// TIA Portal V17 export
// export: Created 2023-02-26T22:53:27.9284899Z, ExportSetting WithDefaults, DisplayName Totally Integrated Automation Portal, DisplayVersion V17, DisplayName TIA Portal Openness, DisplayVersion V17, DisplayName TIA Portal Version Control Interface, DisplayVersion V17, DisplayName TIA Portal Test Suite Advanced, DisplayVersion V17, DisplayName STEP 7 Professional, DisplayVersion V17, DisplayName SIMATIC Energy Suite, DisplayVersion V17, DisplayName STEP 7 Safety, DisplayVersion V17, DisplayName WinCC Professional, DisplayVersion V17
FUNCTION_BLOCK "ERR_LostPackage"   // FB12, LAD
TITLE = Lost Package - Sequential algorithm
{ S7_Optimized_Access := 'TRUE' }
VERSION : 0.1
// stored: AutoNumber true, IsIECCheckEnabled false, IsRetainMemResEnabled false, MemoryReserve 100, SetENOAutomatically false, UDAEnableTagReadback false
   VAR_INPUT
      StartLine : Bool;
      StopLine : Bool;
      AutoMode : Bool;
      ResetButton : Bool;
      Di : Bool;
      Dj : Bool;
      FirstScan : Bool;
      "Time" : Time;
   END_VAR
   VAR_OUTPUT
      Error : Bool;
   END_VAR
   VAR
      S1 : Bool;
      S2 : Bool;
      S3 : Bool;
      t1 : Bool;
      P_ResetButton : Bool;
      IEC_Timer_0_Instance { ExternalAccessible := 'False'; ExternalVisible := 'False'; ExternalWritable := 'False'} : TON_TIME;
   END_VAR
   VAR_TEMP   // added for the SCL form of the ladder/FBD networks
      _w1 : Bool;
   END_VAR
BEGIN

REGION Network 1: Step 3-1
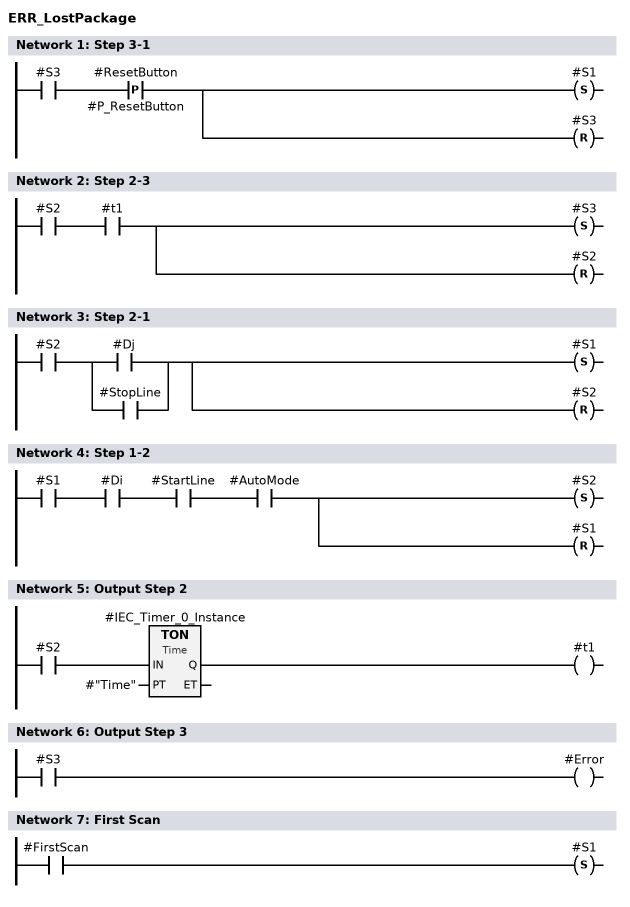
   RUNG wire#powerrail
      Contact( #S3 )
      P_Contact(operand := #ResetButton, bit := #P_ResetButton)
      wire#w1
      S_Coil( #S1 )
   END_RUNG
   RUNG wire#w1
      R_Coil( #S3 )
   END_RUNG
   // the same network as SCL:
   #_w1 := #S3 AND #ResetButton AND NOT #P_ResetButton;   // rising edge of #ResetButton
   #P_ResetButton := #ResetButton;
   IF #_w1 THEN
       #S1 := TRUE;
       #S3 := FALSE;
   END_IF;
END_REGION

REGION Network 2: Step 2-3
   RUNG wire#powerrail
      Contact( #S2 )
      Contact( #t1 )
      wire#w1
      S_Coil( #S3 )
   END_RUNG
   RUNG wire#w1
      R_Coil( #S2 )
   END_RUNG
   // the same network as SCL:
   IF #S2 AND #t1 THEN
       #S3 := TRUE;
       #S2 := FALSE;
   END_IF;
END_REGION

REGION Network 3: Step 2-1
   RUNG wire#powerrail
      Contact( #S2 )
      wire#w1
      Contact( #Dj )
      wire#w2
      S_Coil( #S1 )
   END_RUNG
   RUNG wire#w1
      Contact( #StopLine )
   END_RUNG wire#w2
   RUNG wire#w2
      R_Coil( #S2 )
   END_RUNG
   // the same network as SCL:
   IF #S2 AND (#Dj OR #StopLine) THEN
       #S1 := TRUE;
       #S2 := FALSE;
   END_IF;
END_REGION

REGION Network 4: Step 1-2
   RUNG wire#powerrail
      Contact( #S1 )
      Contact( #Di )
      Contact( #StartLine )
      Contact( #AutoMode )
      wire#w1
      S_Coil( #S2 )
   END_RUNG
   RUNG wire#w1
      R_Coil( #S1 )
   END_RUNG
   // the same network as SCL:
   IF #S1 AND #Di AND #StartLine AND #AutoMode THEN
       #S2 := TRUE;
       #S1 := FALSE;
   END_IF;
END_REGION

REGION Network 5: Output Step 2
   RUNG wire#powerrail
      Contact( #S2 )
      { S7_Templates := "time_type := Time" } #IEC_Timer_0_Instance.TON(pt := #"Time", et =>)
      Coil( #t1 )
   END_RUNG
   // the same network as SCL:
   #IEC_Timer_0_Instance(IN := #S2, PT := #"Time");   // TON
   #t1 := #IEC_Timer_0_Instance.Q;
END_REGION

REGION Network 6: Output Step 3
   RUNG wire#powerrail
      Contact( #S3 )
      Coil( #Error )
   END_RUNG
   // the same network as SCL:
   #Error := #S3;
END_REGION

REGION Network 7: First Scan
   RUNG wire#powerrail
      Contact( #FirstScan )
      S_Coil( #S1 )
   END_RUNG
   // the same network as SCL:
   IF #FirstScan THEN #S1 := TRUE; END_IF;
END_REGION
END_FUNCTION_BLOCK
